FUNCTION_BLOCK FB_AC_Siemens EXTENDS FB_AirConditionerBase
VAR_INPUT
END_VAR
VAR_OUTPUT
END_VAR
VAR
END_VAR

METHOD Execute : BOOL
VAR_INPUT
END_VAR
VAR
	TurnOnCommand: BOOL;
	TurnOffCommand: BOOL;
END_VAR
PublishDeviceData();
END_METHOD

METHOD HandleMessage : BOOL
VAR_INPUT
	message: STRING;
END_VAR
VAR
	TurnOnCommand: BOOL;
	TurnOffCommand: BOOL;
END_VAR
IF TurnOffCommand THEN
	TurnOff();
ELSIF TurnOnCommand THEN
	TurnOn();
END_IF
END_METHOD

METHOD PublishDeviceData : BOOL
VAR_INPUT
END_VAR
END_METHOD

METHOD TurnOff : BOOL
VAR_INPUT
END_VAR
END_METHOD

METHOD TurnOn : BOOL
VAR_INPUT
END_VAR
//turn on Struct created
END_METHOD

END_FUNCTION_BLOCK

(* stored: Version 1.1.0.1, ProductVersion 3.1.4024.9
   POU FB_AC_Siemens: Id {2be6e881-c616-476b-83e6-44913f6addf2}, SpecialFunc None
   Method Execute: Id {f82cfefe-230e-41a1-b485-e0ada534c4a2}
   Method HandleMessage: Id {684407c3-d795-44f4-9757-8aff5132b802}
   Method PublishDeviceData: Id {3ad1dc14-ef6f-4924-9dad-d013aa7b6f38}
   Method TurnOff: Id {248872b0-c69a-479c-be6f-000d0614fdb8}
   Method TurnOn: Id {e5beaa9f-4fbb-4f3b-a7ed-57c55260dc86} *)
